{attribute 'GeneratedUsingTerminal: CU1123-0000-0016'}
{attribute addProperty BoxType "CU1123-0000-0016"}
{attribute addProperty Id "A_0002_CU1123_0010_0016A_0002_CU1123_0010_0016_E68B3D99124"}
{attribute addProperty CRC "820062412"}
{attribute addProperty Size "124"}
{attribute addProperty Name "A_0001(CU1123-0000-0016)"}
TYPE A_0001_CU1123_0000_0016_30E128CC EXTENDS CU1123_1FC0878B :
STRUCT
	{attribute addProperty Name "A_0002(CU1123-0010-0016)"}
	{attribute addProperty PreviousPort "A_0001(CU1123-0000-0016) : D"}
	A_0002_CU1123_0010_0016 : A_0002_CU1123_0010_0016_E68B3D99;
END_STRUCT
END_TYPE

(* stored: Version 1.2.0.0, ProductVersion 3.1.4024.11
   DUT A_0001_CU1123_0000_0016_30E128CC: Id {5e2a46b5-cb0c-48fa-8b5a-1e2547e77942} *)
